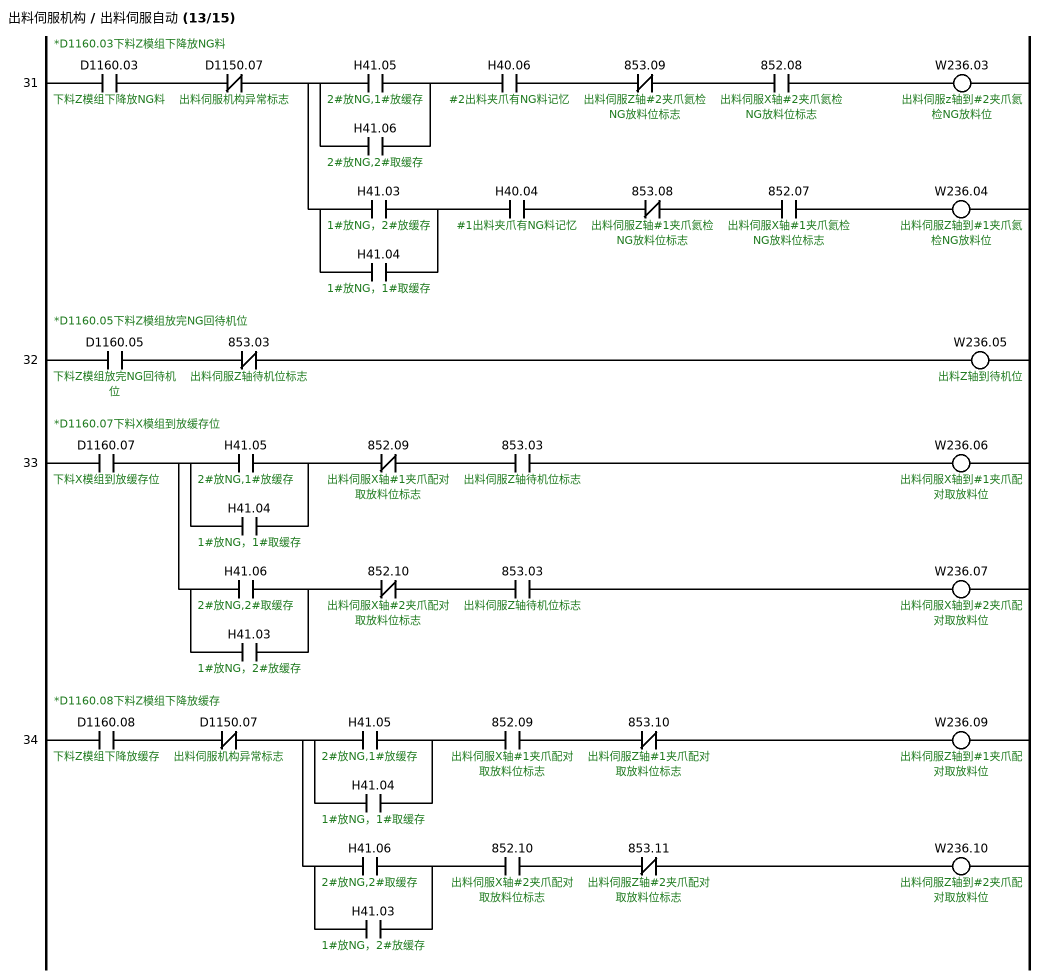
; [picture p456: 出料伺服机构 / 出料伺服自动, rungs 31-34]
; rung 31: *D1160.03下料Z模组下降放NG料
LD D1160.03  ; 下料Z模组下降放NG料
ANDNOT D1150.07  ; 出料伺服机构异常标志
OUT TR0
LD H41.05  ; 2#放NG,1#放缓存
OR H41.06  ; 2#放NG,2#取缓存
ANDLD
AND H40.06  ; #2出料夹爪有NG料记忆
ANDNOT 853.09  ; 出料伺服Z轴#2夹爪氦检NG放料位标志
AND 852.08  ; 出料伺服X轴#2夹爪氦检NG放料位标志
OUT W236.03  ; 出料伺服z轴到#2夹爪氦检NG放料位
LD TR0
LD H41.03  ; 1#放NG，2#放缓存
OR H41.04  ; 1#放NG，1#取缓存
ANDLD
AND H40.04  ; #1出料夹爪有NG料记忆
ANDNOT 853.08  ; 出料伺服Z轴#1夹爪氦检NG放料位标志
AND 852.07  ; 出料伺服X轴#1夹爪氦检NG放料位标志
OUT W236.04  ; 出料伺服Z轴到#1夹爪氦检NG放料位
; rung 32: *D1160.05下料Z模组放完NG回待机位
LD D1160.05  ; 下料Z模组放完NG回待机位
ANDNOT 853.03  ; 出料伺服Z轴待机位标志
OUT W236.05  ; 出料Z轴到待机位
; rung 33: *D1160.07下料X模组到放缓存位
LD D1160.07  ; 下料X模组到放缓存位
OUT TR0
LD H41.05  ; 2#放NG,1#放缓存
OR H41.04  ; 1#放NG，1#取缓存
ANDLD
ANDNOT 852.09  ; 出料伺服X轴#1夹爪配对取放料位标志
AND 853.03  ; 出料伺服Z轴待机位标志
OUT W236.06  ; 出料伺服X轴到#1夹爪配对取放料位
LD TR0
LD H41.06  ; 2#放NG,2#取缓存
OR H41.03  ; 1#放NG，2#放缓存
ANDLD
ANDNOT 852.10  ; 出料伺服X轴#2夹爪配对取放料位标志
AND 853.03  ; 出料伺服Z轴待机位标志
OUT W236.07  ; 出料伺服X轴到#2夹爪配对取放料位
; rung 34: *D1160.08下料Z模组下降放缓存
LD D1160.08  ; 下料Z模组下降放缓存
ANDNOT D1150.07  ; 出料伺服机构异常标志
OUT TR0
LD H41.05  ; 2#放NG,1#放缓存
OR H41.04  ; 1#放NG，1#取缓存
ANDLD
AND 852.09  ; 出料伺服X轴#1夹爪配对取放料位标志
ANDNOT 853.10  ; 出料伺服Z轴#1夹爪配对取放料位标志
OUT W236.09  ; 出料伺服Z轴到#1夹爪配对取放料位
LD TR0
LD H41.06  ; 2#放NG,2#取缓存
OR H41.03  ; 1#放NG，2#放缓存
ANDLD
AND 852.10  ; 出料伺服X轴#2夹爪配对取放料位标志
ANDNOT 853.11  ; 出料伺服Z轴#2夹爪配对取放料位标志
OUT W236.10  ; 出料伺服Z轴到#2夹爪配对取放料位

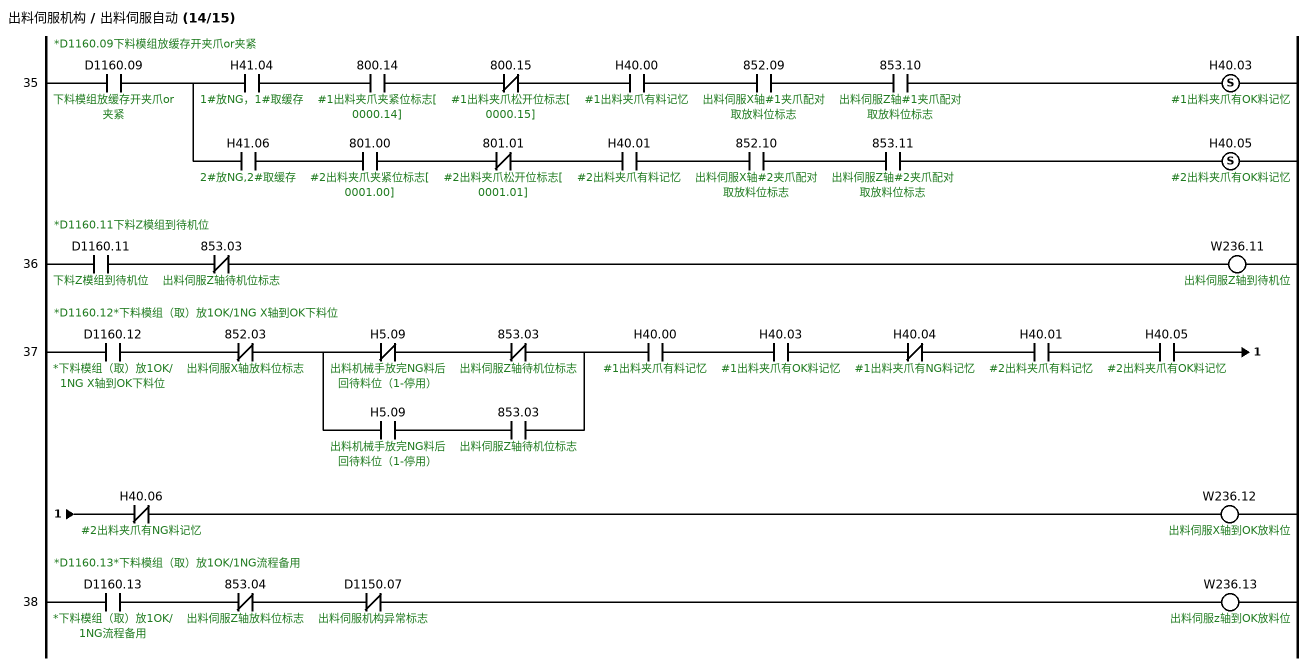
; rung 35: *D1160.09下料模组放缓存开夹爪or夹紧
LD D1160.09  ; 下料模组放缓存开夹爪or夹紧
OUT TR0
AND H41.04  ; 1#放NG，1#取缓存
AND 800.14  ; #1出料夹爪夹紧位标志[0000.14]
ANDNOT 800.15  ; #1出料夹爪松开位标志[0000.15]
AND H40.00  ; #1出料夹爪有料记忆
AND 852.09  ; 出料伺服X轴#1夹爪配对取放料位标志
AND 853.10  ; 出料伺服Z轴#1夹爪配对取放料位标志
SET H40.03  ; #1出料夹爪有OK料记忆
LD TR0
AND H41.06  ; 2#放NG,2#取缓存
AND 801.00  ; #2出料夹爪夹紧位标志[0001.00]
ANDNOT 801.01  ; #2出料夹爪松开位标志[0001.01]
AND H40.01  ; #2出料夹爪有料记忆
AND 852.10  ; 出料伺服X轴#2夹爪配对取放料位标志
AND 853.11  ; 出料伺服Z轴#2夹爪配对取放料位标志
SET H40.05  ; #2出料夹爪有OK料记忆
; rung 36: *D1160.11下料Z模组到待机位
LD D1160.11  ; 下料Z模组到待机位
ANDNOT 853.03  ; 出料伺服Z轴待机位标志
OUT W236.11  ; 出料伺服Z轴到待机位
; rung 37: *D1160.12*下料模组（取）放1OK/1NG X轴到OK下料位
LD D1160.12  ; *下料模组（取）放1OK/1NG X轴到OK下料位
ANDNOT 852.03  ; 出料伺服X轴放料位标志
LDNOT H5.09  ; 出料机械手放完NG料后回待料位（1-停用）
ANDNOT 853.03  ; 出料伺服Z轴待机位标志  // X轴移动条件必须是Z轴在安全位（20190417）
LD H5.09  ; 出料机械手放完NG料后回待料位（1-停用）
AND 853.03  ; 出料伺服Z轴待机位标志
ORLD
ANDLD
AND H40.00  ; #1出料夹爪有料记忆
AND H40.03  ; #1出料夹爪有OK料记忆
ANDNOT H40.04  ; #1出料夹爪有NG料记忆
AND H40.01  ; #2出料夹爪有料记忆
AND H40.05  ; #2出料夹爪有OK料记忆
ANDNOT H40.06  ; #2出料夹爪有NG料记忆
OUT W236.12  ; 出料伺服X轴到OK放料位
; rung 38: *D1160.13*下料模组（取）放1OK/1NG流程备用
LD D1160.13  ; *下料模组（取）放1OK/1NG流程备用
ANDNOT 853.04  ; 出料伺服Z轴放料位标志
ANDNOT D1150.07  ; 出料伺服机构异常标志
OUT W236.13  ; 出料伺服z轴到OK放料位

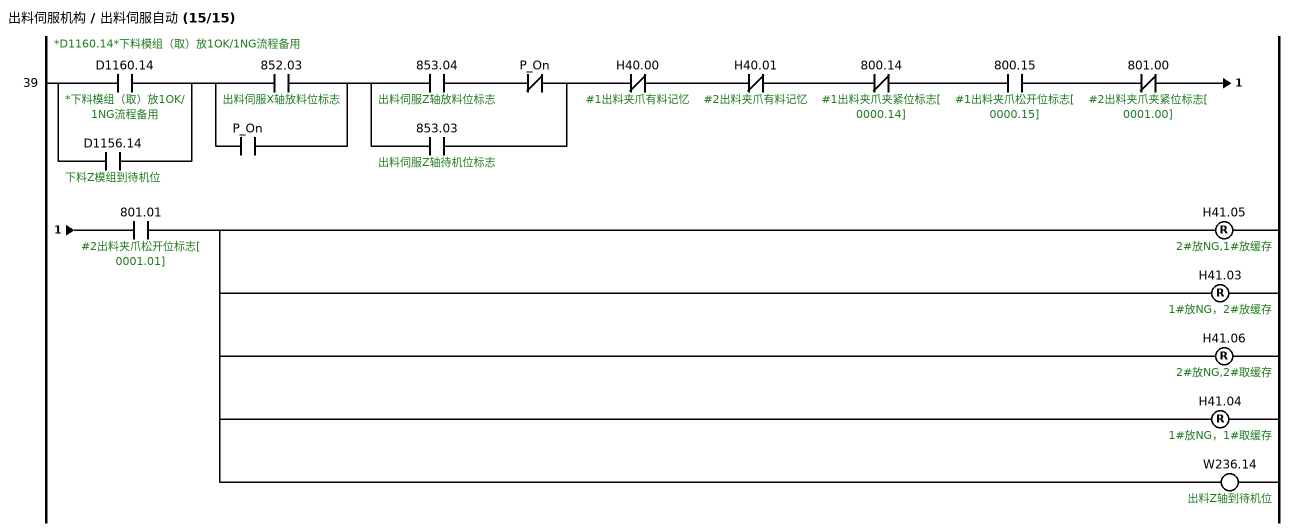
; rung 39: *D1160.14*下料模组（取）放1OK/1NG流程备用
LD D1160.14  ; *下料模组（取）放1OK/1NG流程备用
OR D1156.14  ; 下料Z模组到待机位
LD 852.03  ; 出料伺服X轴放料位标志
OR P_On
ANDLD
LD 853.04  ; 出料伺服Z轴放料位标志
ANDNOT P_On
OR 853.03  ; 出料伺服Z轴待机位标志
ANDLD
ANDNOT H40.00  ; #1出料夹爪有料记忆
ANDNOT H40.01  ; #2出料夹爪有料记忆
ANDNOT 800.14  ; #1出料夹爪夹紧位标志[0000.14]
AND 800.15  ; #1出料夹爪松开位标志[0000.15]
ANDNOT 801.00  ; #2出料夹爪夹紧位标志[0001.00]
AND 801.01  ; #2出料夹爪松开位标志[0001.01]
RSET H41.05  ; 2#放NG,1#放缓存
RSET H41.03  ; 1#放NG，2#放缓存
RSET H41.06  ; 2#放NG,2#取缓存
RSET H41.04  ; 1#放NG，1#取缓存
OUT W236.14  ; 出料Z轴到待机位

### Section 工站复位

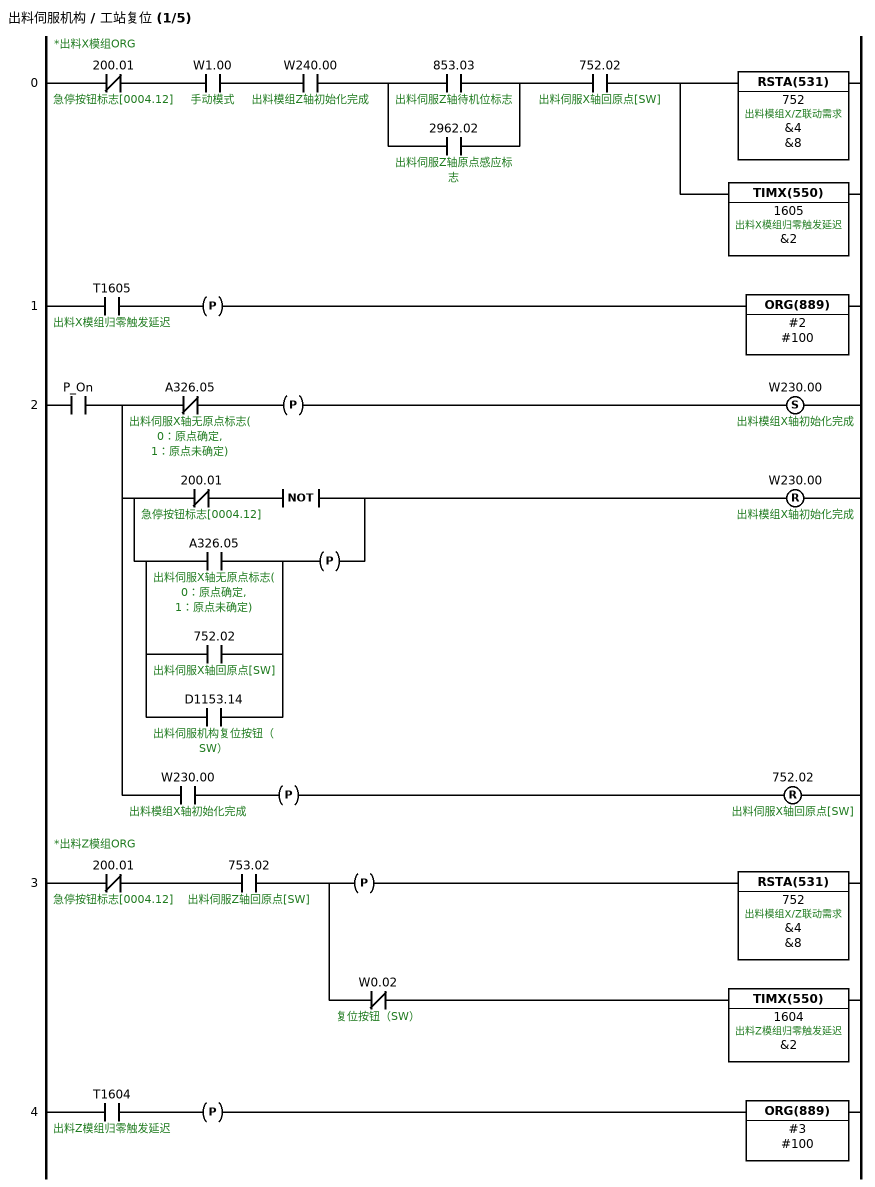
; rung 0: *出料X模组ORG
LDNOT 200.01  ; 急停按钮标志[0004.12]
AND W1.00  ; 手动模式
AND W240.00  ; 出料模组Z轴初始化完成
LD 853.03  ; 出料伺服Z轴待机位标志
OR 2962.02  ; 出料伺服Z轴原点感应标志
ANDLD
AND 752.02  ; 出料伺服X轴回原点[SW]
RSTA(531) 752 &4 &8  ; 出料模组X/Z联动需求
TIMX(550) 1605 &2  ; 出料X模组归零触发延迟
; rung 1
LD T1605  ; 出料X模组归零触发延迟
UP(521)
ORG(889) #2 #100
; rung 2
LD P_On
OUT TR0
ANDNOT A326.05  ; 出料伺服X轴无原点标志(0：原点确定,1：原点未确定)
UP(521)
SET W230.00  ; 出料模组X轴初始化完成
LD TR0
LDNOT 200.01  ; 急停按钮标志[0004.12]
NOT(520)
LD A326.05  ; 出料伺服X轴无原点标志(0：原点确定,1：原点未确定)
OR 752.02  ; 出料伺服X轴回原点[SW]
OR D1153.14  ; 出料伺服机构复位按钮（SW）
UP(521)
ORLD
ANDLD
RSET W230.00  ; 出料模组X轴初始化完成
LD TR0
AND W230.00  ; 出料模组X轴初始化完成
UP(521)
RSET 752.02  ; 出料伺服X轴回原点[SW]
; rung 3: *出料Z模组ORG
LDNOT 200.01  ; 急停按钮标志[0004.12]
AND 753.02  ; 出料伺服Z轴回原点[SW]
OUT TR0
UP(521)
RSTA(531) 752 &4 &8  ; 出料模组X/Z联动需求
LD TR0
ANDNOT W0.02  ; 复位按钮（SW）
TIMX(550) 1604 &2  ; 出料Z模组归零触发延迟
; rung 4
LD T1604  ; 出料Z模组归零触发延迟
UP(521)
ORG(889) #3 #100

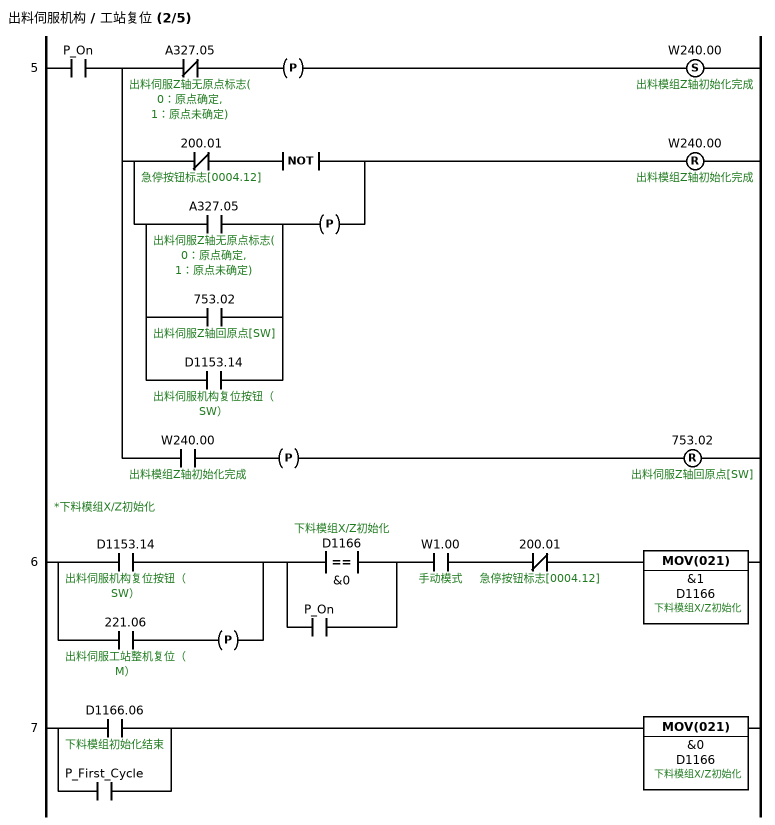
; rung 5
LD P_On
OUT TR0
ANDNOT A327.05  ; 出料伺服Z轴无原点标志(0：原点确定,1：原点未确定)
UP(521)
SET W240.00  ; 出料模组Z轴初始化完成
LD TR0
LDNOT 200.01  ; 急停按钮标志[0004.12]
NOT(520)
LD A327.05  ; 出料伺服Z轴无原点标志(0：原点确定,1：原点未确定)
OR 753.02  ; 出料伺服Z轴回原点[SW]
OR D1153.14  ; 出料伺服机构复位按钮（SW）
UP(521)
ORLD
ANDLD
RSET W240.00  ; 出料模组Z轴初始化完成
LD TR0
AND W240.00  ; 出料模组Z轴初始化完成
UP(521)
RSET 753.02  ; 出料伺服Z轴回原点[SW]
; rung 6: *下料模组X/Z初始化
LD D1153.14  ; 出料伺服机构复位按钮（SW）
LD 221.06  ; 出料伺服工站整机复位（M）
UP(521)
ORLD
LD=(300) D1166 &0  ; 下料模组X/Z初始化
OR P_On
ANDLD
AND W1.00  ; 手动模式
ANDNOT 200.01  ; 急停按钮标志[0004.12]
MOV(021) &1 D1166  ; 下料模组X/Z初始化
; rung 7
LD D1166.06  ; 下料模组初始化结束
OR P_First_Cycle
MOV(021) &0 D1166  ; 下料模组X/Z初始化

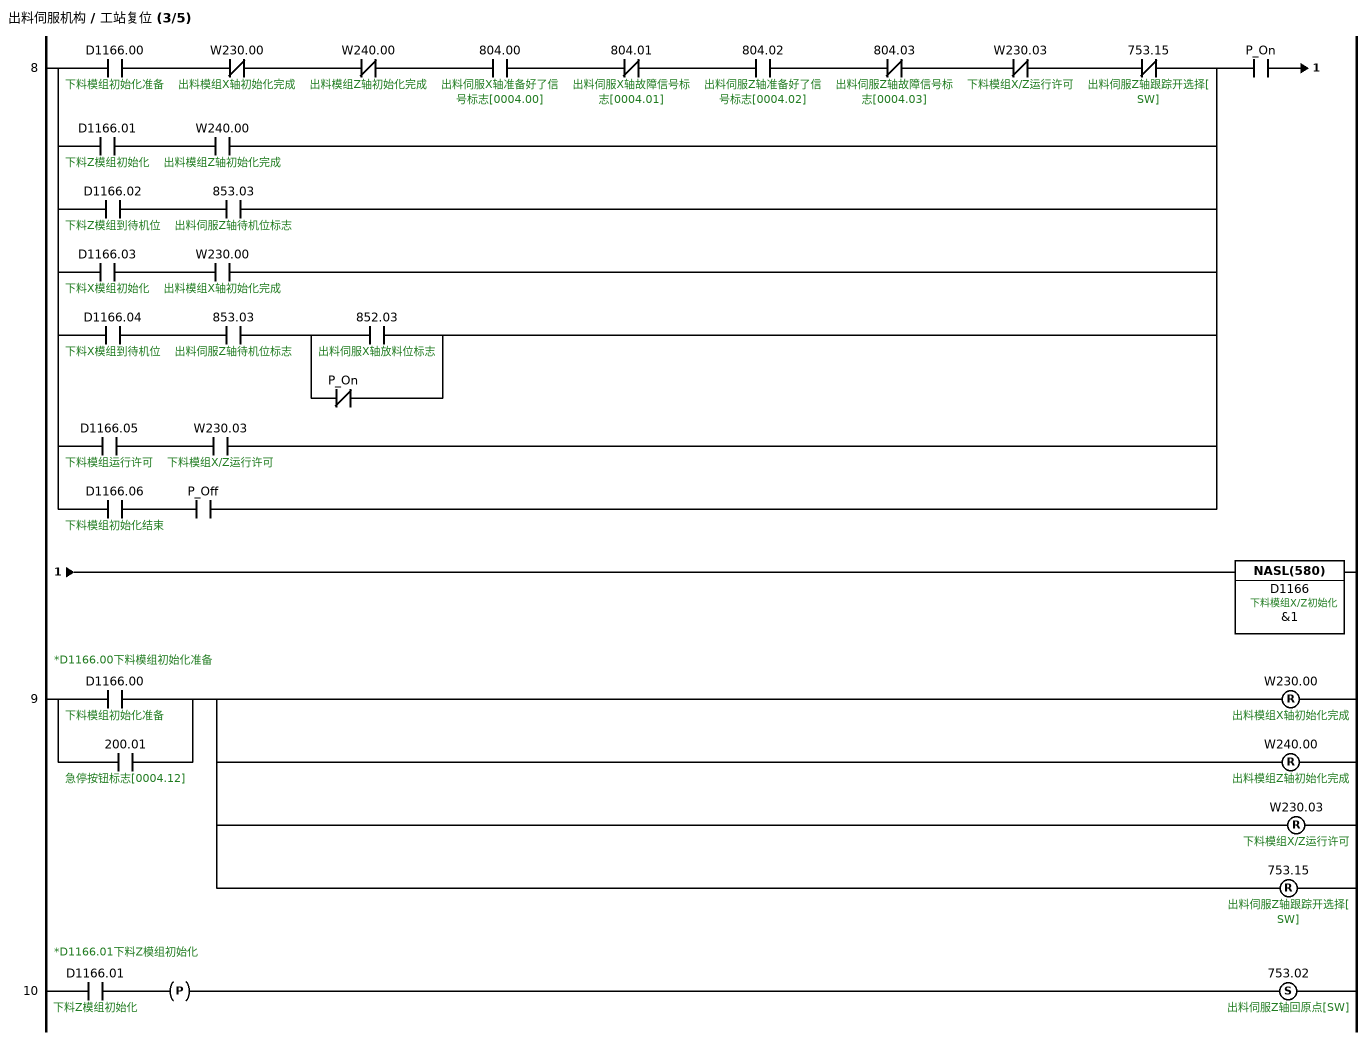
; rung 8
LD D1166.00  ; 下料模组初始化准备
ANDNOT W230.00  ; 出料模组X轴初始化完成
ANDNOT W240.00  ; 出料模组Z轴初始化完成
AND 804.00  ; 出料伺服X轴准备好了信号标志[0004.00]
ANDNOT 804.01  ; 出料伺服X轴故障信号标志[0004.01]
AND 804.02  ; 出料伺服Z轴准备好了信号标志[0004.02]
ANDNOT 804.03  ; 出料伺服Z轴故障信号标志[0004.03]
ANDNOT W230.03  ; 下料模组X/Z运行许可
ANDNOT 753.15  ; 出料伺服Z轴跟踪开选择[SW]
LD D1166.01  ; 下料Z模组初始化
AND W240.00  ; 出料模组Z轴初始化完成
ORLD
LD D1166.02  ; 下料Z模组到待机位
AND 853.03  ; 出料伺服Z轴待机位标志
ORLD
LD D1166.03  ; 下料X模组初始化
AND W230.00  ; 出料模组X轴初始化完成
ORLD
LD D1166.04  ; 下料X模组到待机位
AND 853.03  ; 出料伺服Z轴待机位标志
LD 852.03  ; 出料伺服X轴放料位标志
ORNOT P_On
ANDLD
ORLD
LD D1166.05  ; 下料模组运行许可
AND W230.03  ; 下料模组X/Z运行许可
ORLD
LD D1166.06  ; 下料模组初始化结束
AND P_Off
ORLD
AND P_On
NASL(580) D1166 &1  ; 下料模组X/Z初始化
; rung 9: *D1166.00下料模组初始化准备
LD D1166.00  ; 下料模组初始化准备
OR 200.01  ; 急停按钮标志[0004.12]
RSET W230.00  ; 出料模组X轴初始化完成
RSET W240.00  ; 出料模组Z轴初始化完成
RSET W230.03  ; 下料模组X/Z运行许可
RSET 753.15  ; 出料伺服Z轴跟踪开选择[SW]
; rung 10: *D1166.01下料Z模组初始化
LD D1166.01  ; 下料Z模组初始化
UP(521)
SET 753.02  ; 出料伺服Z轴回原点[SW]

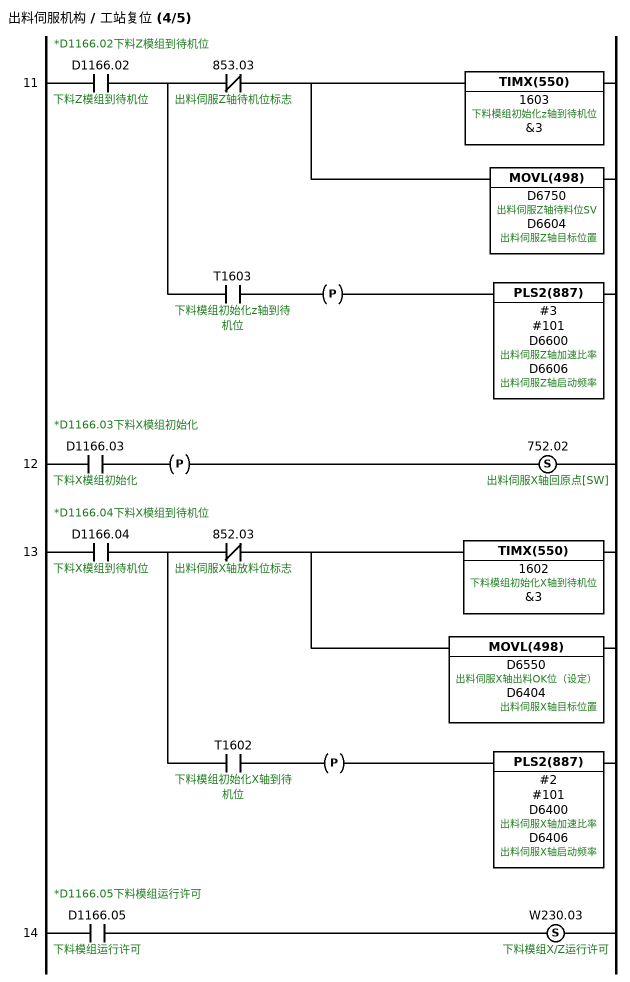
; rung 11: *D1166.02下料Z模组到待机位
LD D1166.02  ; 下料Z模组到待机位
OUT TR0
ANDNOT 853.03  ; 出料伺服Z轴待机位标志
TIMX(550) 1603 &3  ; 下料模组初始化z轴到待机位
MOVL(498) D6750 D6604  ; 出料伺服Z轴待料位SV, 出料伺服Z轴目标位置
LD TR0
AND T1603  ; 下料模组初始化z轴到待机位
UP(521)
PLS2(887) #3 #101 D6600 D6606  ; 出料伺服Z轴加速比率, 出料伺服Z轴启动频率
; rung 12: *D1166.03下料X模组初始化
LD D1166.03  ; 下料X模组初始化
UP(521)
SET 752.02  ; 出料伺服X轴回原点[SW]
; rung 13: *D1166.04下料X模组到待机位
LD D1166.04  ; 下料X模组到待机位
OUT TR0
ANDNOT 852.03  ; 出料伺服X轴放料位标志
TIMX(550) 1602 &3  ; 下料模组初始化X轴到待机位
MOVL(498) D6550 D6404  ; 出料伺服X轴出料OK位（设定）, 出料伺服X轴目标位置
LD TR0
AND T1602  ; 下料模组初始化X轴到待机位
UP(521)
PLS2(887) #2 #101 D6400 D6406  ; 出料伺服X轴加速比率, 出料伺服X轴启动频率
; rung 14: *D1166.05下料模组运行许可
LD D1166.05  ; 下料模组运行许可
SET W230.03  ; 下料模组X/Z运行许可

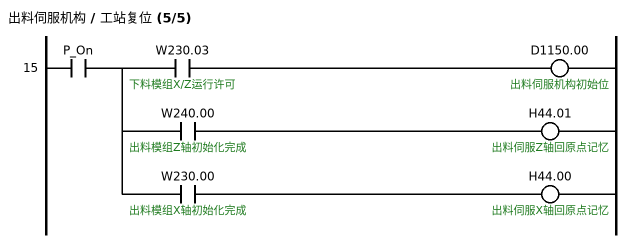
; rung 15
LD P_On
OUT TR0
AND W230.03  ; 下料模组X/Z运行许可
OUT D1150.00  ; 出料伺服机构初始位
LD TR0
AND W240.00  ; 出料模组Z轴初始化完成
OUT H44.01  ; 出料伺服Z轴回原点记忆
LD TR0
AND W230.00  ; 出料模组X轴初始化完成
OUT H44.00  ; 出料伺服X轴回原点记忆

### Section 指示灯

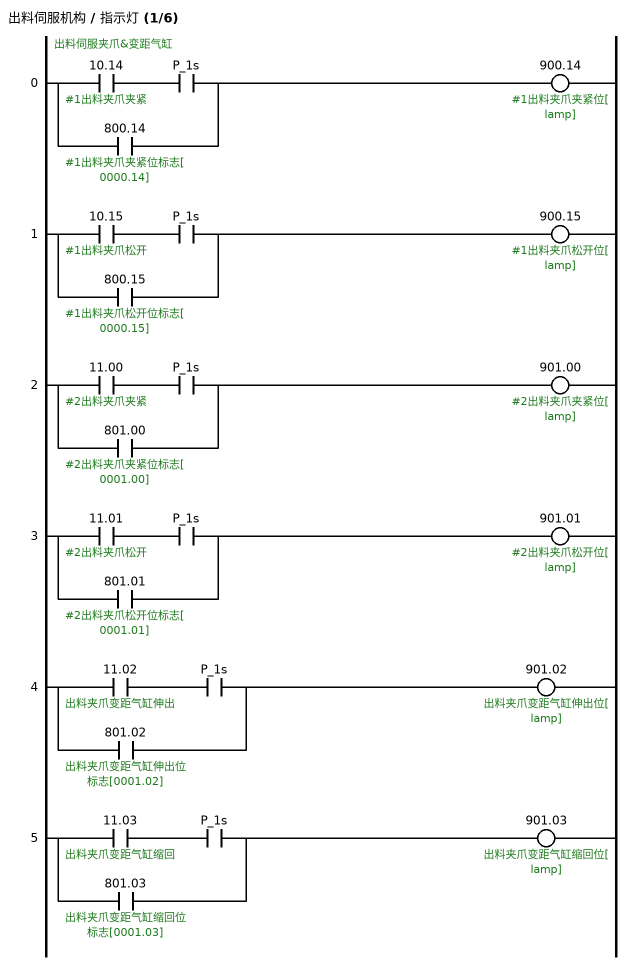
; rung 0: 出料伺服夹爪&变距气缸
LD 10.14  ; #1出料夹爪夹紧
AND P_1s
OR 800.14  ; #1出料夹爪夹紧位标志[0000.14]
OUT 900.14  ; #1出料夹爪夹紧位[lamp]
; rung 1
LD 10.15  ; #1出料夹爪松开
AND P_1s
OR 800.15  ; #1出料夹爪松开位标志[0000.15]
OUT 900.15  ; #1出料夹爪松开位[lamp]
; rung 2
LD 11.00  ; #2出料夹爪夹紧
AND P_1s
OR 801.00  ; #2出料夹爪夹紧位标志[0001.00]
OUT 901.00  ; #2出料夹爪夹紧位[lamp]
; rung 3
LD 11.01  ; #2出料夹爪松开
AND P_1s
OR 801.01  ; #2出料夹爪松开位标志[0001.01]
OUT 901.01  ; #2出料夹爪松开位[lamp]
; rung 4
LD 11.02  ; 出料夹爪变距气缸伸出
AND P_1s
OR 801.02  ; 出料夹爪变距气缸伸出位标志[0001.02]
OUT 901.02  ; 出料夹爪变距气缸伸出位[lamp]
; rung 5
LD 11.03  ; 出料夹爪变距气缸缩回
AND P_1s
OR 801.03  ; 出料夹爪变距气缸缩回位标志[0001.03]
OUT 901.03  ; 出料夹爪变距气缸缩回位[lamp]

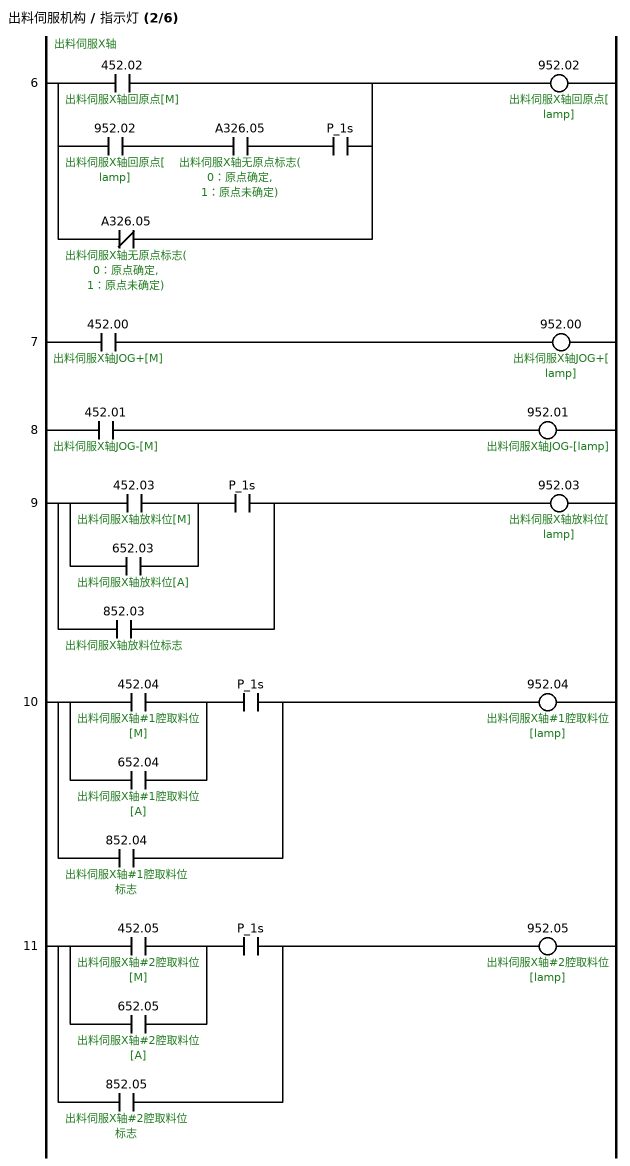
; rung 6: 出料伺服X轴
LD 452.02  ; 出料伺服X轴回原点[M]
LD 952.02  ; 出料伺服X轴回原点[lamp]
AND A326.05  ; 出料伺服X轴无原点标志(0：原点确定,1：原点未确定)
AND P_1s
ORLD
ORNOT A326.05  ; 出料伺服X轴无原点标志(0：原点确定,1：原点未确定)
OUT 952.02  ; 出料伺服X轴回原点[lamp]
; rung 7
LD 452.00  ; 出料伺服X轴JOG+[M]
OUT 952.00  ; 出料伺服X轴JOG+[lamp]
; rung 8
LD 452.01  ; 出料伺服X轴JOG-[M]
OUT 952.01  ; 出料伺服X轴JOG-[lamp]
; rung 9
LD 452.03  ; 出料伺服X轴放料位[M]
OR 652.03  ; 出料伺服X轴放料位[A]
AND P_1s
OR 852.03  ; 出料伺服X轴放料位标志
OUT 952.03  ; 出料伺服X轴放料位[lamp]
; rung 10
LD 452.04  ; 出料伺服X轴#1腔取料位[M]
OR 652.04  ; 出料伺服X轴#1腔取料位[A]
AND P_1s
OR 852.04  ; 出料伺服X轴#1腔取料位标志
OUT 952.04  ; 出料伺服X轴#1腔取料位[lamp]
; rung 11
LD 452.05  ; 出料伺服X轴#2腔取料位[M]
OR 652.05  ; 出料伺服X轴#2腔取料位[A]
AND P_1s
OR 852.05  ; 出料伺服X轴#2腔取料位标志
OUT 952.05  ; 出料伺服X轴#2腔取料位[lamp]

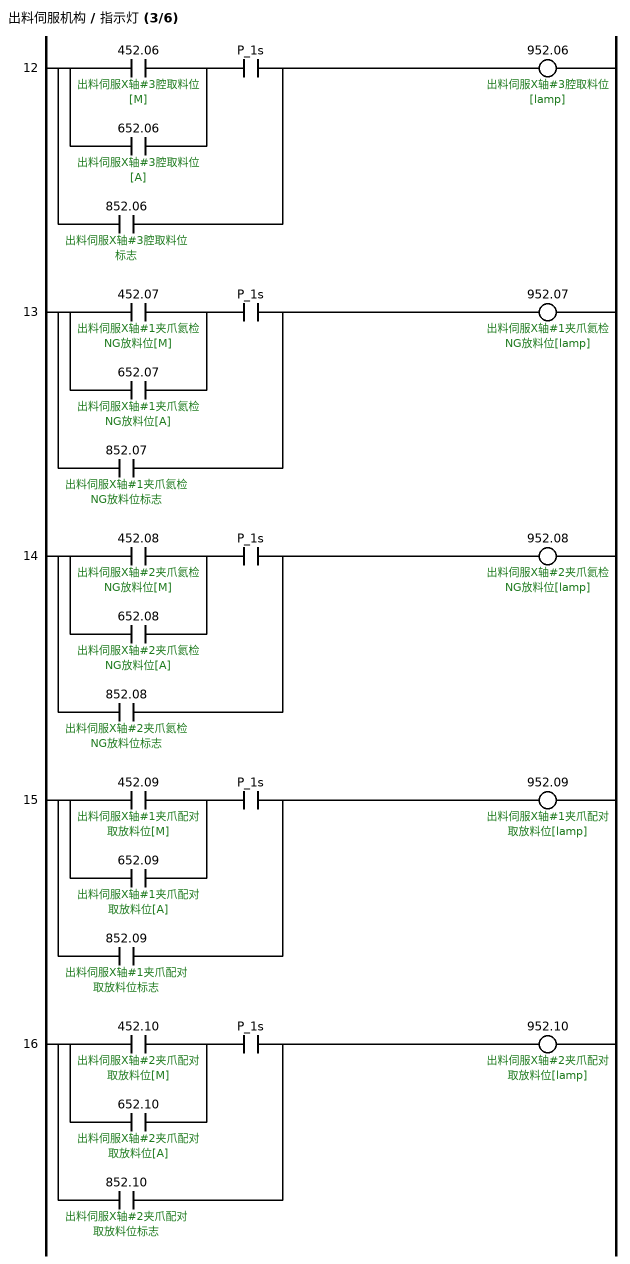
; rung 12
LD 452.06  ; 出料伺服X轴#3腔取料位[M]
OR 652.06  ; 出料伺服X轴#3腔取料位[A]
AND P_1s
OR 852.06  ; 出料伺服X轴#3腔取料位标志
OUT 952.06  ; 出料伺服X轴#3腔取料位[lamp]
; rung 13
LD 452.07  ; 出料伺服X轴#1夹爪氦检NG放料位[M]
OR 652.07  ; 出料伺服X轴#1夹爪氦检NG放料位[A]
AND P_1s
OR 852.07  ; 出料伺服X轴#1夹爪氦检NG放料位标志
OUT 952.07  ; 出料伺服X轴#1夹爪氦检NG放料位[lamp]
; rung 14
LD 452.08  ; 出料伺服X轴#2夹爪氦检NG放料位[M]
OR 652.08  ; 出料伺服X轴#2夹爪氦检NG放料位[A]
AND P_1s
OR 852.08  ; 出料伺服X轴#2夹爪氦检NG放料位标志
OUT 952.08  ; 出料伺服X轴#2夹爪氦检NG放料位[lamp]
; rung 15
LD 452.09  ; 出料伺服X轴#1夹爪配对取放料位[M]
OR 652.09  ; 出料伺服X轴#1夹爪配对取放料位[A]
AND P_1s
OR 852.09  ; 出料伺服X轴#1夹爪配对取放料位标志
OUT 952.09  ; 出料伺服X轴#1夹爪配对取放料位[lamp]
; rung 16
LD 452.10  ; 出料伺服X轴#2夹爪配对取放料位[M]
OR 652.10  ; 出料伺服X轴#2夹爪配对取放料位[A]
AND P_1s
OR 852.10  ; 出料伺服X轴#2夹爪配对取放料位标志
OUT 952.10  ; 出料伺服X轴#2夹爪配对取放料位[lamp]

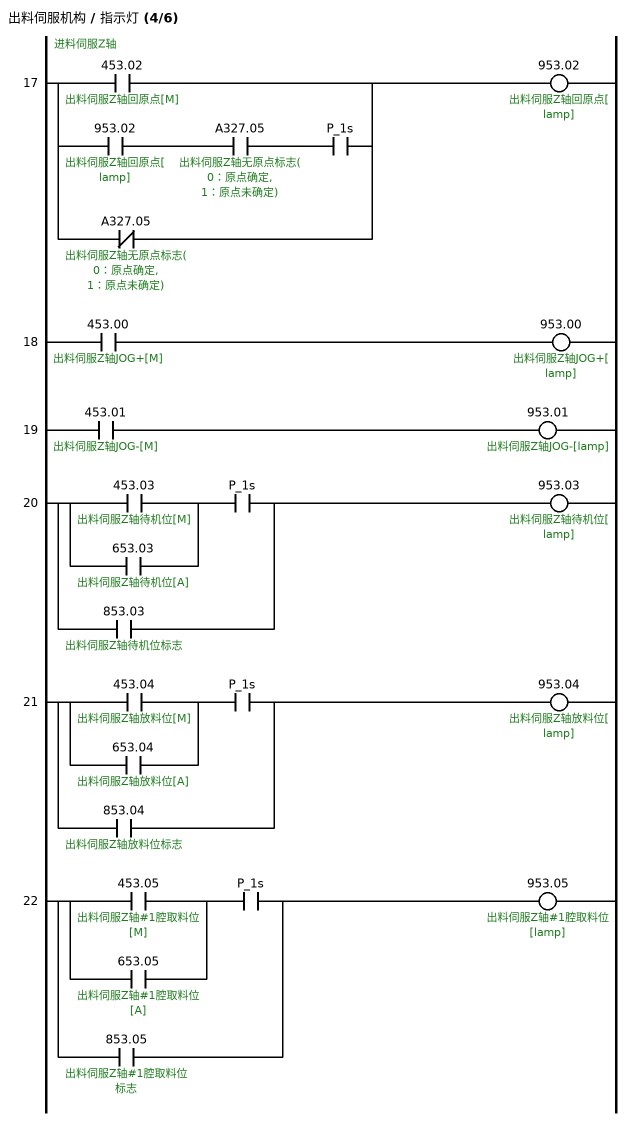
; rung 17: 进料伺服Z轴
LD 453.02  ; 出料伺服Z轴回原点[M]
LD 953.02  ; 出料伺服Z轴回原点[lamp]
AND A327.05  ; 出料伺服Z轴无原点标志(0：原点确定,1：原点未确定)
AND P_1s
ORLD
ORNOT A327.05  ; 出料伺服Z轴无原点标志(0：原点确定,1：原点未确定)
OUT 953.02  ; 出料伺服Z轴回原点[lamp]
; rung 18
LD 453.00  ; 出料伺服Z轴JOG+[M]
OUT 953.00  ; 出料伺服Z轴JOG+[lamp]
; rung 19
LD 453.01  ; 出料伺服Z轴JOG-[M]
OUT 953.01  ; 出料伺服Z轴JOG-[lamp]
; rung 20
LD 453.03  ; 出料伺服Z轴待机位[M]
OR 653.03  ; 出料伺服Z轴待机位[A]
AND P_1s
OR 853.03  ; 出料伺服Z轴待机位标志
OUT 953.03  ; 出料伺服Z轴待机位[lamp]
; rung 21
LD 453.04  ; 出料伺服Z轴放料位[M]
OR 653.04  ; 出料伺服Z轴放料位[A]
AND P_1s
OR 853.04  ; 出料伺服Z轴放料位标志
OUT 953.04  ; 出料伺服Z轴放料位[lamp]
; rung 22
LD 453.05  ; 出料伺服Z轴#1腔取料位[M]
OR 653.05  ; 出料伺服Z轴#1腔取料位[A]
AND P_1s
OR 853.05  ; 出料伺服Z轴#1腔取料位标志
OUT 953.05  ; 出料伺服Z轴#1腔取料位[lamp]

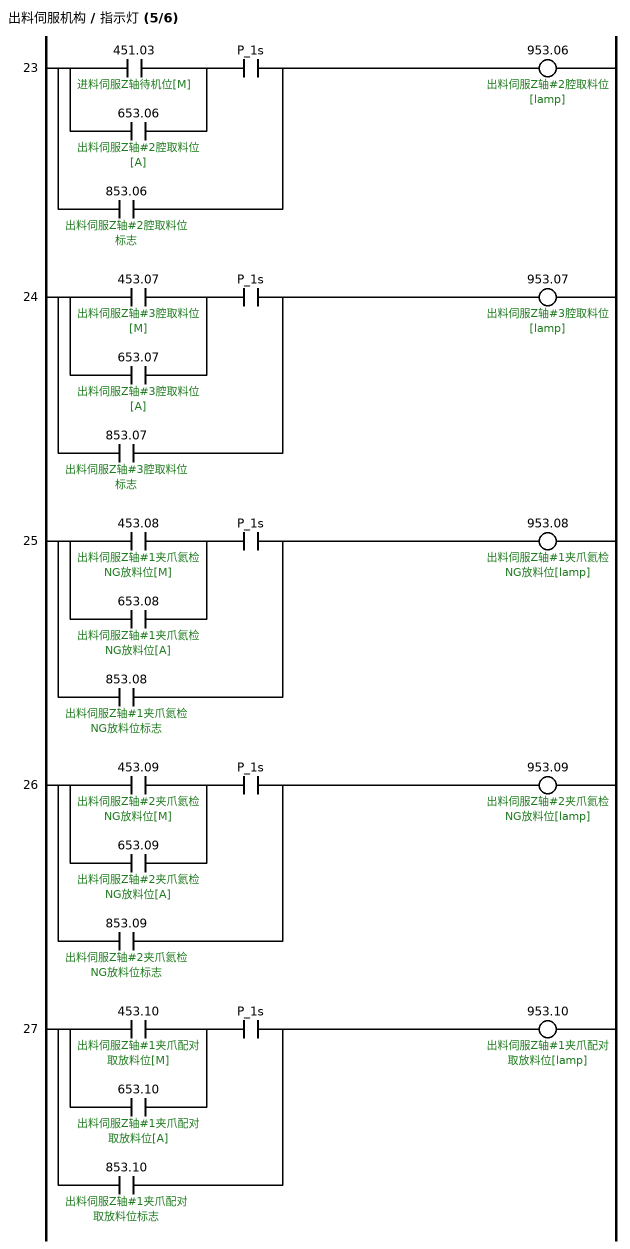
; rung 23
LD 451.03  ; 进料伺服Z轴待机位[M]
OR 653.06  ; 出料伺服Z轴#2腔取料位[A]
AND P_1s
OR 853.06  ; 出料伺服Z轴#2腔取料位标志
OUT 953.06  ; 出料伺服Z轴#2腔取料位[lamp]
; rung 24
LD 453.07  ; 出料伺服Z轴#3腔取料位[M]
OR 653.07  ; 出料伺服Z轴#3腔取料位[A]
AND P_1s
OR 853.07  ; 出料伺服Z轴#3腔取料位标志
OUT 953.07  ; 出料伺服Z轴#3腔取料位[lamp]
; rung 25
LD 453.08  ; 出料伺服Z轴#1夹爪氦检NG放料位[M]
OR 653.08  ; 出料伺服Z轴#1夹爪氦检NG放料位[A]
AND P_1s
OR 853.08  ; 出料伺服Z轴#1夹爪氦检NG放料位标志
OUT 953.08  ; 出料伺服Z轴#1夹爪氦检NG放料位[lamp]
; rung 26
LD 453.09  ; 出料伺服Z轴#2夹爪氦检NG放料位[M]
OR 653.09  ; 出料伺服Z轴#2夹爪氦检NG放料位[A]
AND P_1s
OR 853.09  ; 出料伺服Z轴#2夹爪氦检NG放料位标志
OUT 953.09  ; 出料伺服Z轴#2夹爪氦检NG放料位[lamp]
; rung 27
LD 453.10  ; 出料伺服Z轴#1夹爪配对取放料位[M]
OR 653.10  ; 出料伺服Z轴#1夹爪配对取放料位[A]
AND P_1s
OR 853.10  ; 出料伺服Z轴#1夹爪配对取放料位标志
OUT 953.10  ; 出料伺服Z轴#1夹爪配对取放料位[lamp]

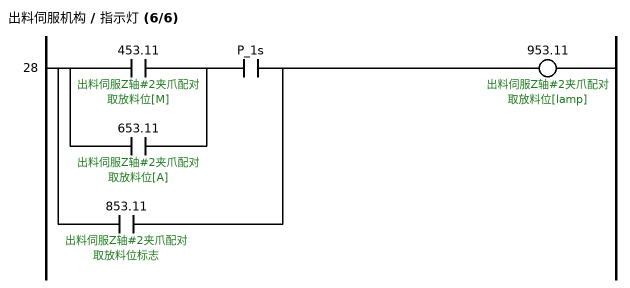
; rung 28
LD 453.11  ; 出料伺服Z轴#2夹爪配对取放料位[M]
OR 653.11  ; 出料伺服Z轴#2夹爪配对取放料位[A]
AND P_1s
OR 853.11  ; 出料伺服Z轴#2夹爪配对取放料位标志
OUT 953.11  ; 出料伺服Z轴#2夹爪配对取放料位[lamp]

### Section 外部输出

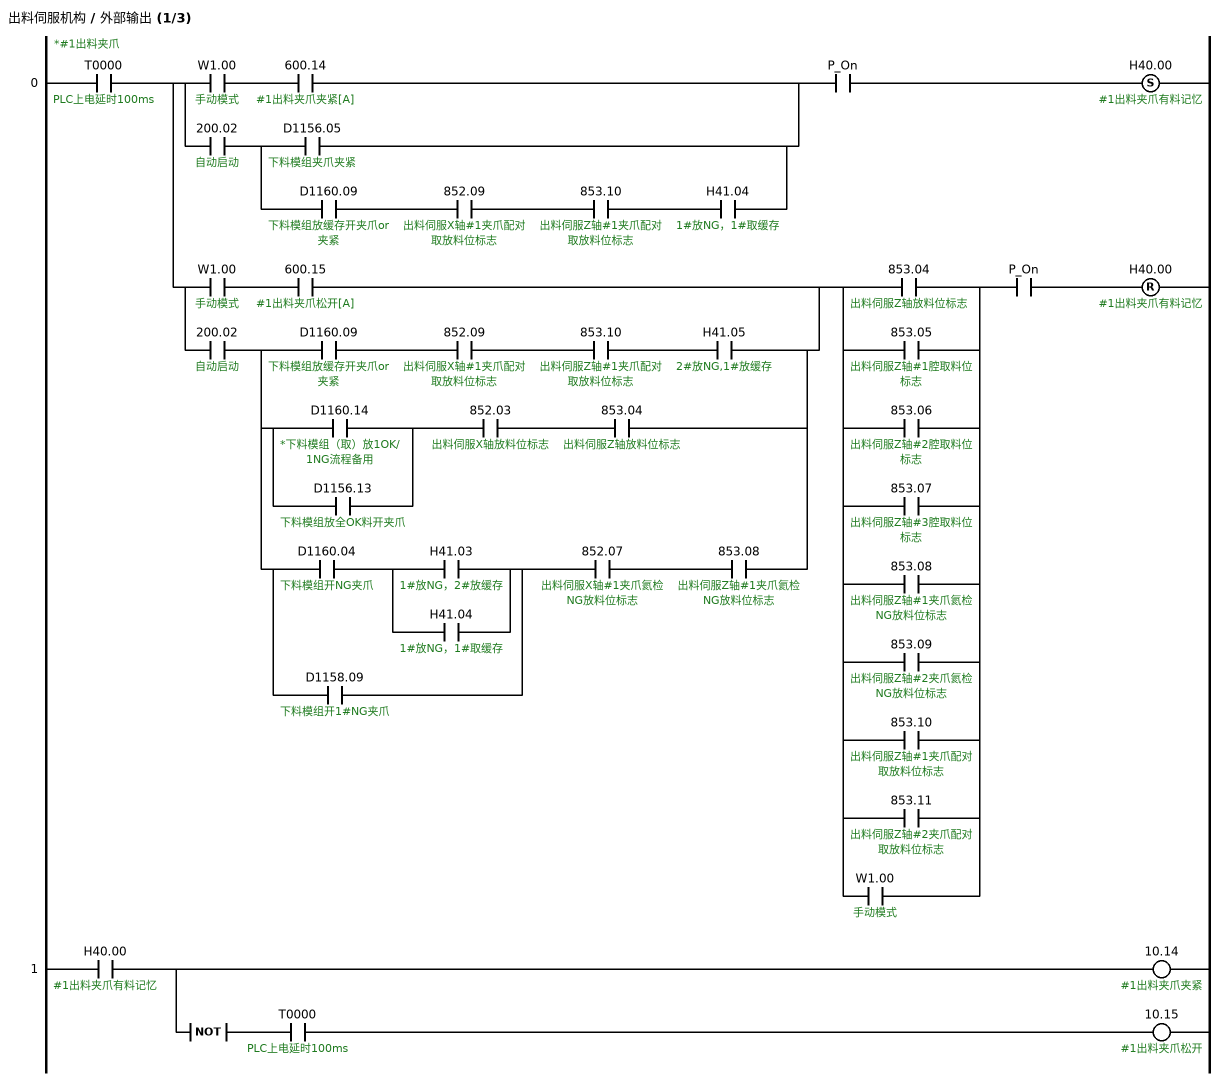
; rung 0: *#1出料夹爪
LD T0000  ; PLC上电延时100ms
OUT TR0
LD W1.00  ; 手动模式
AND 600.14  ; #1出料夹爪夹紧[A]
LD 200.02  ; 自动启动
LD D1156.05  ; 下料模组夹爪夹紧
LD D1160.09  ; 下料模组放缓存开夹爪or夹紧
AND 852.09  ; 出料伺服X轴#1夹爪配对取放料位标志
AND 853.10  ; 出料伺服Z轴#1夹爪配对取放料位标志
AND H41.04  ; 1#放NG，1#取缓存
ORLD
ANDLD
ORLD
ANDLD
AND P_On
SET H40.00  ; #1出料夹爪有料记忆
LD TR0
LD W1.00  ; 手动模式
AND 600.15  ; #1出料夹爪松开[A]
LD 200.02  ; 自动启动
LD D1160.09  ; 下料模组放缓存开夹爪or夹紧
AND 852.09  ; 出料伺服X轴#1夹爪配对取放料位标志
AND 853.10  ; 出料伺服Z轴#1夹爪配对取放料位标志
AND H41.05  ; 2#放NG,1#放缓存
LD D1160.14  ; *下料模组（取）放1OK/1NG流程备用
OR D1156.13  ; 下料模组放全OK料开夹爪
AND 852.03  ; 出料伺服X轴放料位标志
AND 853.04  ; 出料伺服Z轴放料位标志
ORLD
LD D1160.04  ; 下料模组开NG夹爪
LD H41.03  ; 1#放NG，2#放缓存
OR H41.04  ; 1#放NG，1#取缓存
ANDLD
OR D1158.09  ; 下料模组开1#NG夹爪
AND 852.07  ; 出料伺服X轴#1夹爪氦检NG放料位标志
AND 853.08  ; 出料伺服Z轴#1夹爪氦检NG放料位标志
ORLD
ANDLD
ORLD
ANDLD
LD 853.04  ; 出料伺服Z轴放料位标志
OR 853.05  ; 出料伺服Z轴#1腔取料位标志
OR 853.06  ; 出料伺服Z轴#2腔取料位标志
OR 853.07  ; 出料伺服Z轴#3腔取料位标志
OR 853.08  ; 出料伺服Z轴#1夹爪氦检NG放料位标志
OR 853.09  ; 出料伺服Z轴#2夹爪氦检NG放料位标志
OR 853.10  ; 出料伺服Z轴#1夹爪配对取放料位标志
OR 853.11  ; 出料伺服Z轴#2夹爪配对取放料位标志
OR W1.00  ; 手动模式
ANDLD
AND P_On
RSET H40.00  ; #1出料夹爪有料记忆
; rung 1
LD H40.00  ; #1出料夹爪有料记忆
OUT 10.14  ; #1出料夹爪夹紧
NOT(520)
AND T0000  ; PLC上电延时100ms
OUT 10.15  ; #1出料夹爪松开

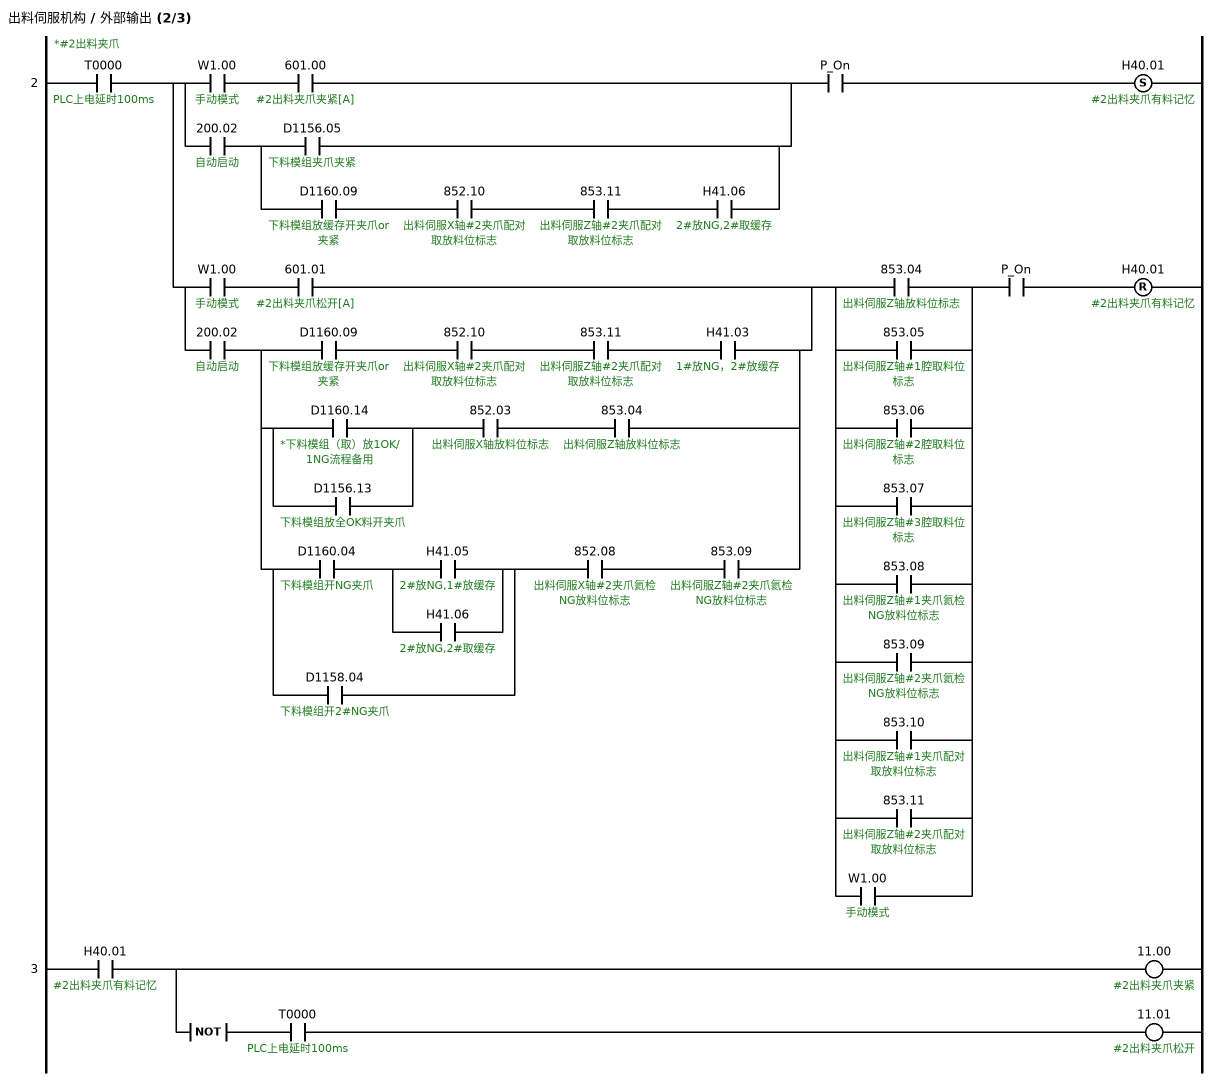
; rung 2: *#2出料夹爪
LD T0000  ; PLC上电延时100ms
OUT TR0
LD W1.00  ; 手动模式
AND 601.00  ; #2出料夹爪夹紧[A]
LD 200.02  ; 自动启动
LD D1156.05  ; 下料模组夹爪夹紧
LD D1160.09  ; 下料模组放缓存开夹爪or夹紧
AND 852.10  ; 出料伺服X轴#2夹爪配对取放料位标志
AND 853.11  ; 出料伺服Z轴#2夹爪配对取放料位标志
AND H41.06  ; 2#放NG,2#取缓存
ORLD
ANDLD
ORLD
ANDLD
AND P_On
SET H40.01  ; #2出料夹爪有料记忆
LD TR0
LD W1.00  ; 手动模式
AND 601.01  ; #2出料夹爪松开[A]
LD 200.02  ; 自动启动
LD D1160.09  ; 下料模组放缓存开夹爪or夹紧
AND 852.10  ; 出料伺服X轴#2夹爪配对取放料位标志
AND 853.11  ; 出料伺服Z轴#2夹爪配对取放料位标志
AND H41.03  ; 1#放NG，2#放缓存
LD D1160.14  ; *下料模组（取）放1OK/1NG流程备用
OR D1156.13  ; 下料模组放全OK料开夹爪
AND 852.03  ; 出料伺服X轴放料位标志
AND 853.04  ; 出料伺服Z轴放料位标志
ORLD
LD D1160.04  ; 下料模组开NG夹爪
LD H41.05  ; 2#放NG,1#放缓存
OR H41.06  ; 2#放NG,2#取缓存
ANDLD
OR D1158.04  ; 下料模组开2#NG夹爪
AND 852.08  ; 出料伺服X轴#2夹爪氦检NG放料位标志
AND 853.09  ; 出料伺服Z轴#2夹爪氦检NG放料位标志
ORLD
ANDLD
ORLD
ANDLD
LD 853.04  ; 出料伺服Z轴放料位标志
OR 853.05  ; 出料伺服Z轴#1腔取料位标志
OR 853.06  ; 出料伺服Z轴#2腔取料位标志
OR 853.07  ; 出料伺服Z轴#3腔取料位标志
OR 853.08  ; 出料伺服Z轴#1夹爪氦检NG放料位标志
OR 853.09  ; 出料伺服Z轴#2夹爪氦检NG放料位标志
OR 853.10  ; 出料伺服Z轴#1夹爪配对取放料位标志
OR 853.11  ; 出料伺服Z轴#2夹爪配对取放料位标志
OR W1.00  ; 手动模式
ANDLD
AND P_On
RSET H40.01  ; #2出料夹爪有料记忆
; rung 3
LD H40.01  ; #2出料夹爪有料记忆
OUT 11.00  ; #2出料夹爪夹紧
NOT(520)
AND T0000  ; PLC上电延时100ms
OUT 11.01  ; #2出料夹爪松开

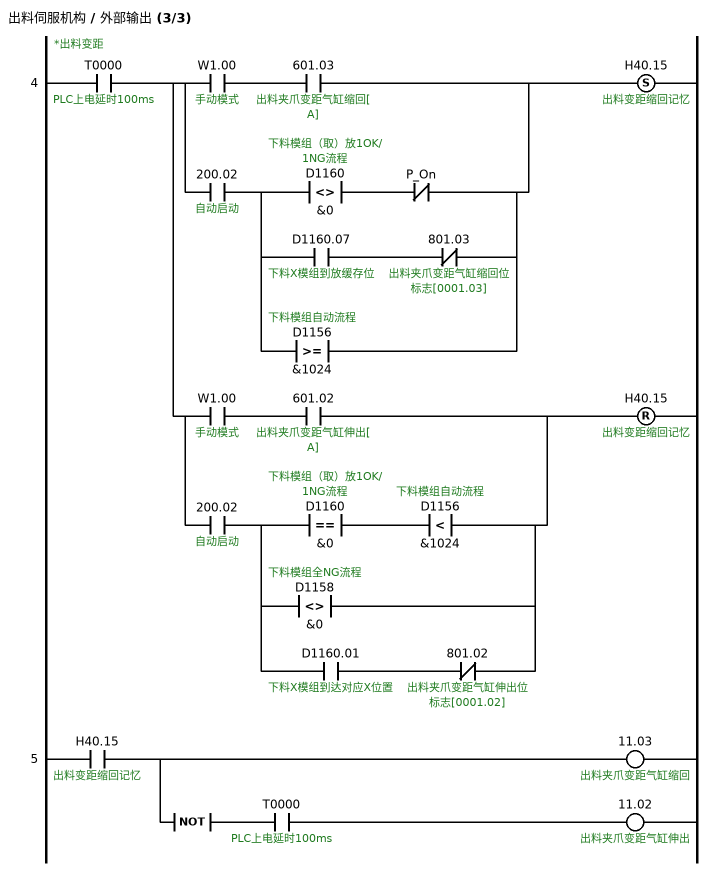
; rung 4: *出料变距
LD T0000  ; PLC上电延时100ms
OUT TR0
LD W1.00  ; 手动模式
AND 601.03  ; 出料夹爪变距气缸缩回[A]
LD 200.02  ; 自动启动
LD<>L(306) D1160 &0  ; 下料模组（取）放1OK/1NG流程
ANDNOT P_On
LD D1160.07  ; 下料X模组到放缓存位
ANDNOT 801.03  ; 出料夹爪变距气缸缩回位标志[0001.03]  // 20190126新增
ORLD
OR>=L(326) D1156 &1024  ; 下料模组自动流程
ANDLD
ORLD
ANDLD
SET H40.15  ; 出料变距缩回记忆
LD TR0
LD W1.00  ; 手动模式
AND 601.02  ; 出料夹爪变距气缸伸出[A]
LD 200.02  ; 自动启动
LD=L(301) D1160 &0  ; 下料模组（取）放1OK/1NG流程
AND<L(311) D1156 &1024  ; 下料模组自动流程
OR<>L(306) D1158 &0  ; 下料模组全NG流程
LD D1160.01  ; 下料X模组到达对应X位置
ANDNOT 801.02  ; 出料夹爪变距气缸伸出位标志[0001.02]  // 20190126新增
ORLD
ANDLD
ORLD
ANDLD
RSET H40.15  ; 出料变距缩回记忆
; rung 5
LD H40.15  ; 出料变距缩回记忆
OUT 11.03  ; 出料夹爪变距气缸缩回
NOT(520)
AND T0000  ; PLC上电延时100ms
OUT 11.02  ; 出料夹爪变距气缸伸出

### Section END
; rung 0
END(001)

## Program NG缓存机构 (cyclic task 5)

### Section NG缓存

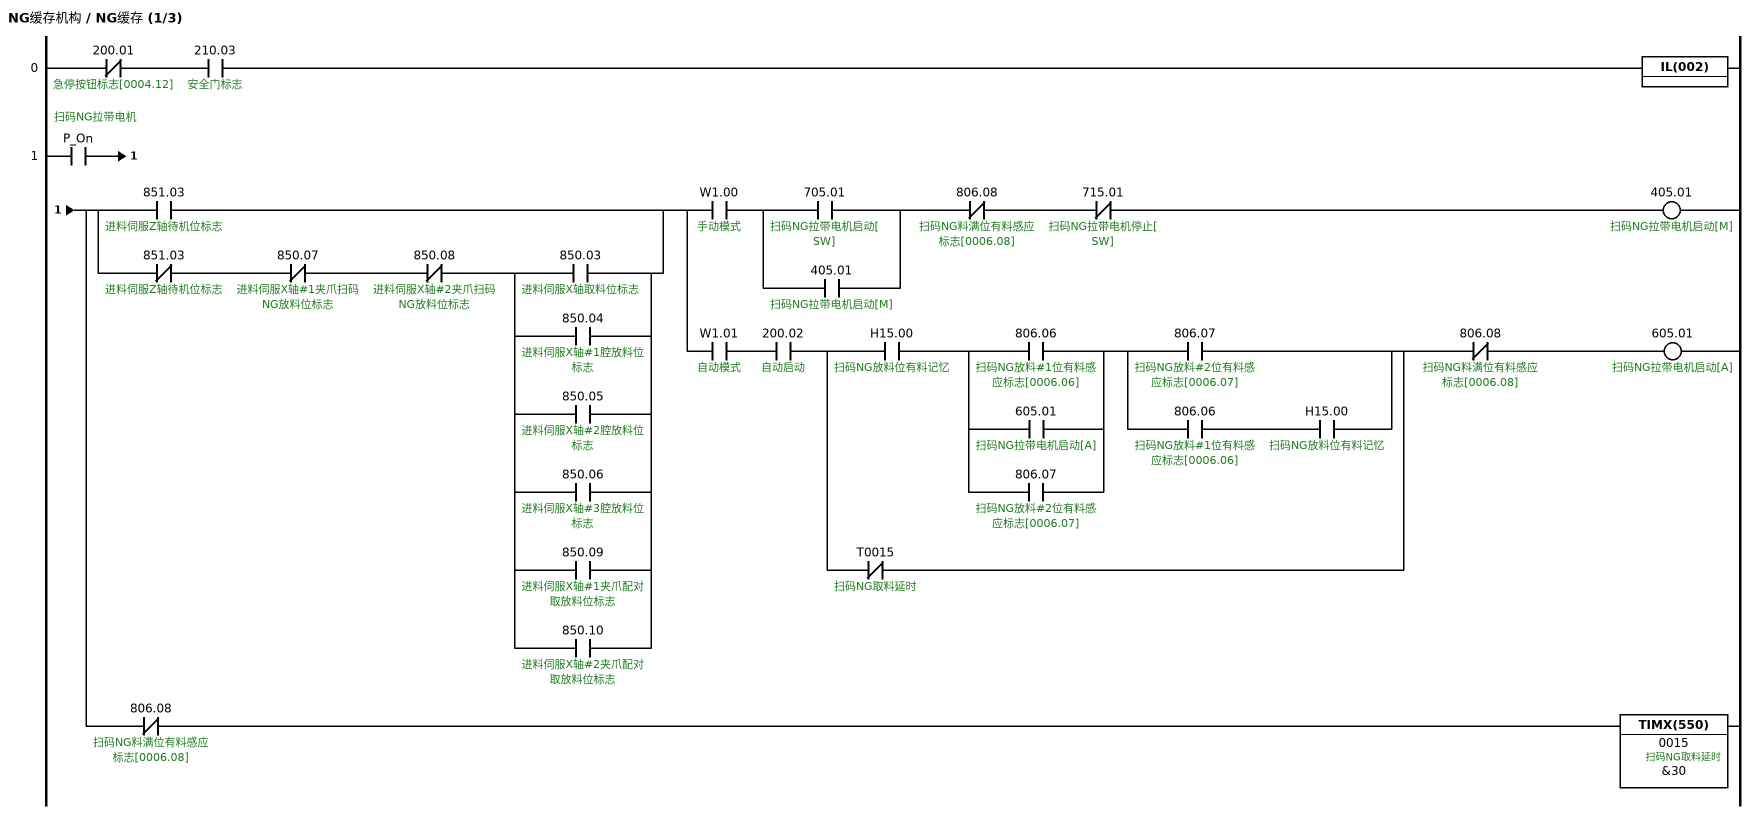
; rung 0
LDNOT 200.01  ; 急停按钮标志[0004.12]
AND 210.03  ; 安全门标志
IL(002)
; rung 1: 扫码NG拉带电机
LD P_On
OUT TR0
LD 851.03  ; 进料伺服Z轴待机位标志
LDNOT 851.03  ; 进料伺服Z轴待机位标志
ANDNOT 850.07  ; 进料伺服X轴#1夹爪扫码NG放料位标志
ANDNOT 850.08  ; 进料伺服X轴#2夹爪扫码NG放料位标志
LD 850.03  ; 进料伺服X轴取料位标志
OR 850.04  ; 进料伺服X轴#1腔放料位标志
OR 850.05  ; 进料伺服X轴#2腔放料位标志
OR 850.06  ; 进料伺服X轴#3腔放料位标志
OR 850.09  ; 进料伺服X轴#1夹爪配对取放料位标志
OR 850.10  ; 进料伺服X轴#2夹爪配对取放料位标志
ANDLD
ORLD
ANDLD
OUT TR1
AND W1.00  ; 手动模式
LD 705.01  ; 扫码NG拉带电机启动[SW]
OR 405.01  ; 扫码NG拉带电机启动[M]
ANDLD
ANDNOT 806.08  ; 扫码NG料满位有料感应标志[0006.08]
ANDNOT 715.01  ; 扫码NG拉带电机停止[SW]
OUT 405.01  ; 扫码NG拉带电机启动[M]
LD TR1
AND W1.01  ; 自动模式
AND 200.02  ; 自动启动
LD H15.00  ; 扫码NG放料位有料记忆
LD 806.06  ; 扫码NG放料#1位有料感应标志[0006.06]
OR 605.01  ; 扫码NG拉带电机启动[A]
OR 806.07  ; 扫码NG放料#2位有料感应标志[0006.07]
ANDLD
LD 806.07  ; 扫码NG放料#2位有料感应标志[0006.07]
LD 806.06  ; 扫码NG放料#1位有料感应标志[0006.06]
AND H15.00  ; 扫码NG放料位有料记忆
ORLD
ANDLD
ORNOT T0015  ; 扫码NG取料延时
ANDLD
ANDNOT 806.08  ; 扫码NG料满位有料感应标志[0006.08]
OUT 605.01  ; 扫码NG拉带电机启动[A]
LD TR0
ANDNOT 806.08  ; 扫码NG料满位有料感应标志[0006.08]
TIMX(550) 0015 &30  ; 扫码NG取料延时

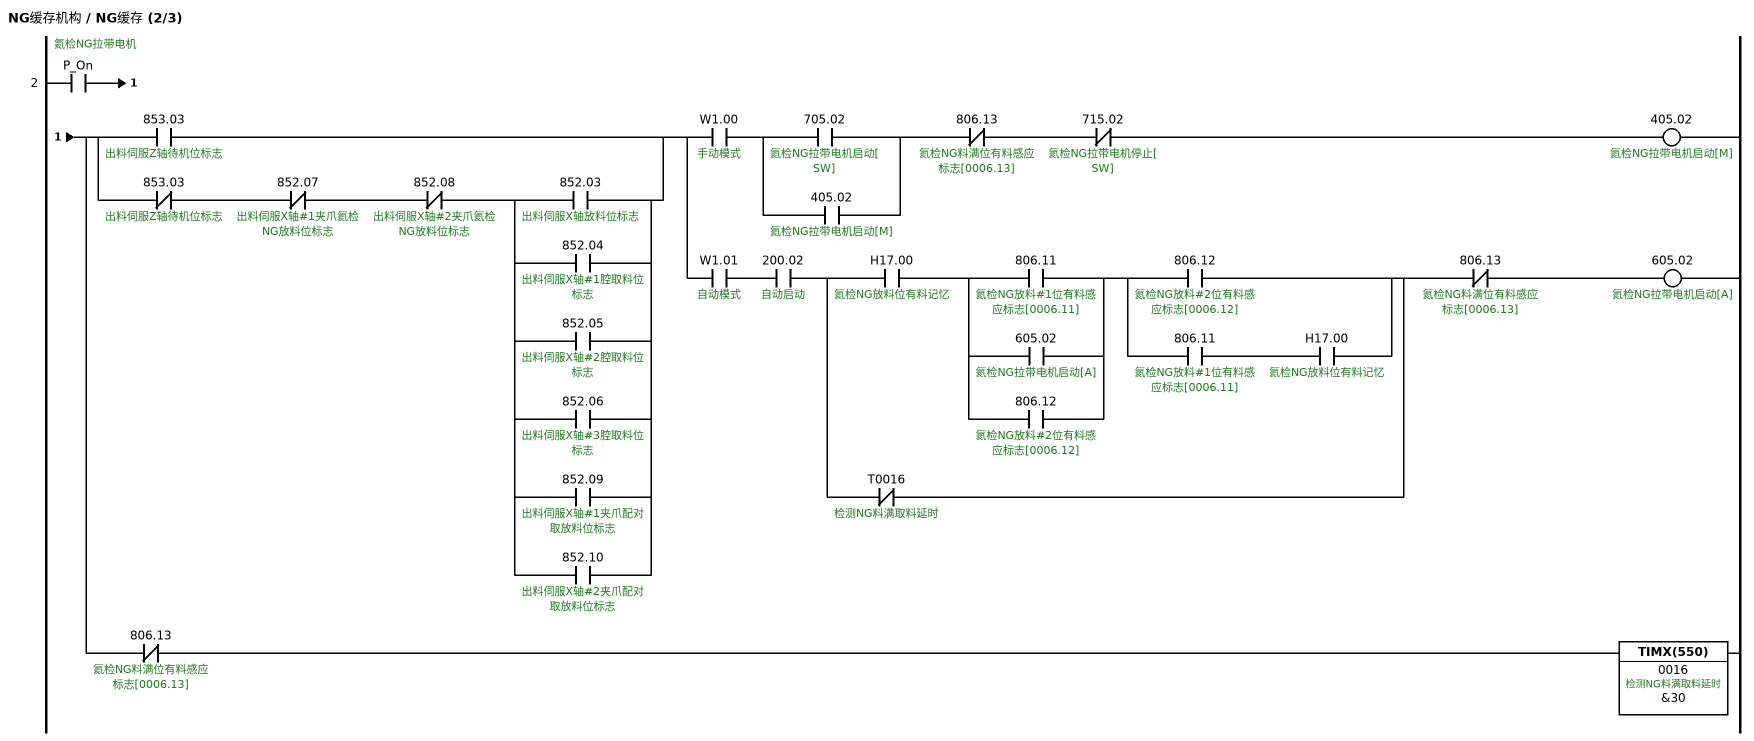
; rung 2: 氦检NG拉带电机
LD P_On
OUT TR0
LD 853.03  ; 出料伺服Z轴待机位标志
LDNOT 853.03  ; 出料伺服Z轴待机位标志
ANDNOT 852.07  ; 出料伺服X轴#1夹爪氦检NG放料位标志
ANDNOT 852.08  ; 出料伺服X轴#2夹爪氦检NG放料位标志
LD 852.03  ; 出料伺服X轴放料位标志
OR 852.04  ; 出料伺服X轴#1腔取料位标志
OR 852.05  ; 出料伺服X轴#2腔取料位标志
OR 852.06  ; 出料伺服X轴#3腔取料位标志
OR 852.09  ; 出料伺服X轴#1夹爪配对取放料位标志
OR 852.10  ; 出料伺服X轴#2夹爪配对取放料位标志
ANDLD
ORLD
ANDLD
OUT TR1
AND W1.00  ; 手动模式
LD 705.02  ; 氦检NG拉带电机启动[SW]
OR 405.02  ; 氦检NG拉带电机启动[M]
ANDLD
ANDNOT 806.13  ; 氦检NG料满位有料感应标志[0006.13]
ANDNOT 715.02  ; 氦检NG拉带电机停止[SW]
OUT 405.02  ; 氦检NG拉带电机启动[M]
LD TR1
AND W1.01  ; 自动模式
AND 200.02  ; 自动启动
LD H17.00  ; 氦检NG放料位有料记忆
LD 806.11  ; 氦检NG放料#1位有料感应标志[0006.11]
OR 605.02  ; 氦检NG拉带电机启动[A]
OR 806.12  ; 氦检NG放料#2位有料感应标志[0006.12]
ANDLD
LD 806.12  ; 氦检NG放料#2位有料感应标志[0006.12]
LD 806.11  ; 氦检NG放料#1位有料感应标志[0006.11]
AND H17.00  ; 氦检NG放料位有料记忆
ORLD
ANDLD
ORNOT T0016  ; 检测NG料满取料延时
ANDLD
ANDNOT 806.13  ; 氦检NG料满位有料感应标志[0006.13]
OUT 605.02  ; 氦检NG拉带电机启动[A]
LD TR0
ANDNOT 806.13  ; 氦检NG料满位有料感应标志[0006.13]
TIMX(550) 0016 &30  ; 检测NG料满取料延时

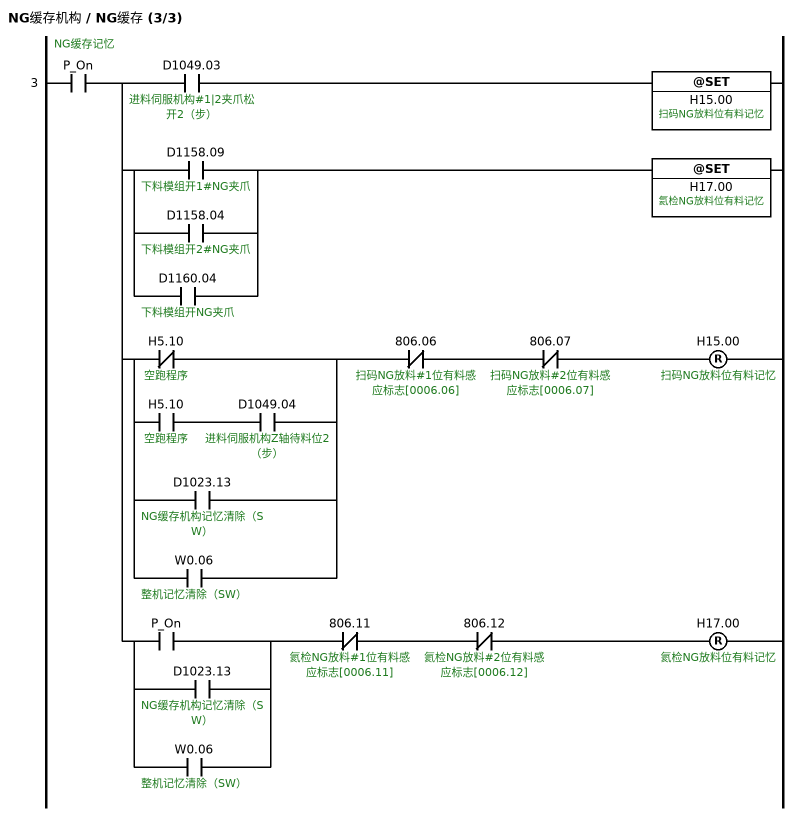
; rung 3: NG缓存记忆
LD P_On
OUT TR0
AND D1049.03  ; 进料伺服机构#1|2夹爪松开2（步）
@SET H15.00  ; 扫码NG放料位有料记忆
LD TR0
LD D1158.09  ; 下料模组开1#NG夹爪
OR D1158.04  ; 下料模组开2#NG夹爪
OR D1160.04  ; 下料模组开NG夹爪
ANDLD
@SET H17.00  ; 氦检NG放料位有料记忆
LD TR0
LDNOT H5.10  ; 空跑程序
LD H5.10  ; 空跑程序
AND D1049.04  ; 进料伺服机构Z轴待料位2（步）
ORLD
OR D1023.13  ; NG缓存机构记忆清除（SW）
OR W0.06  ; 整机记忆清除（SW）
ANDLD
ANDNOT 806.06  ; 扫码NG放料#1位有料感应标志[0006.06]
ANDNOT 806.07  ; 扫码NG放料#2位有料感应标志[0006.07]
RSET H15.00  ; 扫码NG放料位有料记忆
LD TR0
LD P_On
OR D1023.13  ; NG缓存机构记忆清除（SW）
OR W0.06  ; 整机记忆清除（SW）
ANDLD
ANDNOT 806.11  ; 氦检NG放料#1位有料感应标志[0006.11]
ANDNOT 806.12  ; 氦检NG放料#2位有料感应标志[0006.12]
RSET H17.00  ; 氦检NG放料位有料记忆

### Section 外部输出

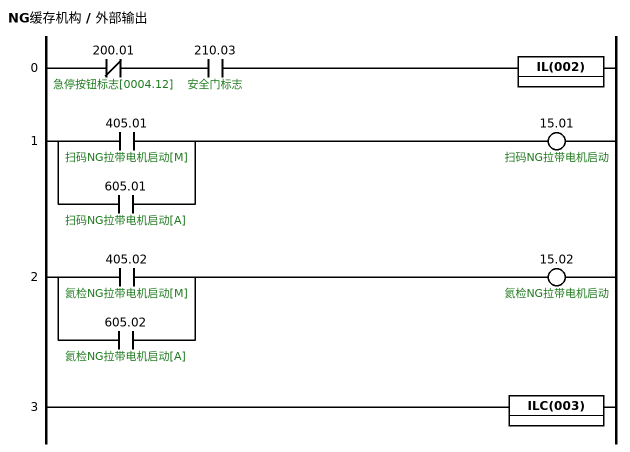
; rung 0
LDNOT 200.01  ; 急停按钮标志[0004.12]
AND 210.03  ; 安全门标志
IL(002)
; rung 1
LD 405.01  ; 扫码NG拉带电机启动[M]
OR 605.01  ; 扫码NG拉带电机启动[A]
OUT 15.01  ; 扫码NG拉带电机启动
; rung 2
LD 405.02  ; 氦检NG拉带电机启动[M]
OR 605.02  ; 氦检NG拉带电机启动[A]
OUT 15.02  ; 氦检NG拉带电机启动
; rung 3
ILC(003)

### Section END
; rung 0
END(001)

## Program Common (cyclic task 6)

### Section 动作延时

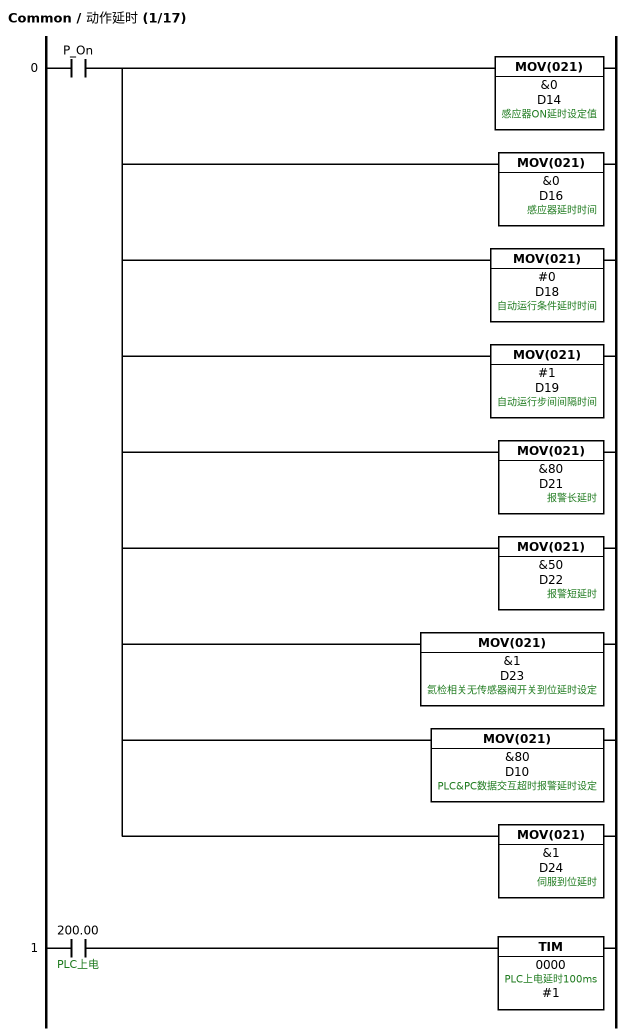
; rung 0
LD P_On
MOV(021) &0 D14  ; 感应器ON延时设定值
MOV(021) &0 D16  ; 感应器延时时间
MOV(021) #0 D18  ; 自动运行条件延时时间
MOV(021) #1 D19  ; 自动运行步间间隔时间
MOV(021) &80 D21  ; 报警长延时
MOV(021) &50 D22  ; 报警短延时
MOV(021) &1 D23  ; 氦检相关无传感器阀开关到位延时设定
MOV(021) &80 D10  ; PLC&PC数据交互超时报警延时设定
MOV(021) &1 D24  ; 伺服到位延时
; rung 1
LD 200.00  ; PLC上电
TIM 0000 #1  ; PLC上电延时100ms

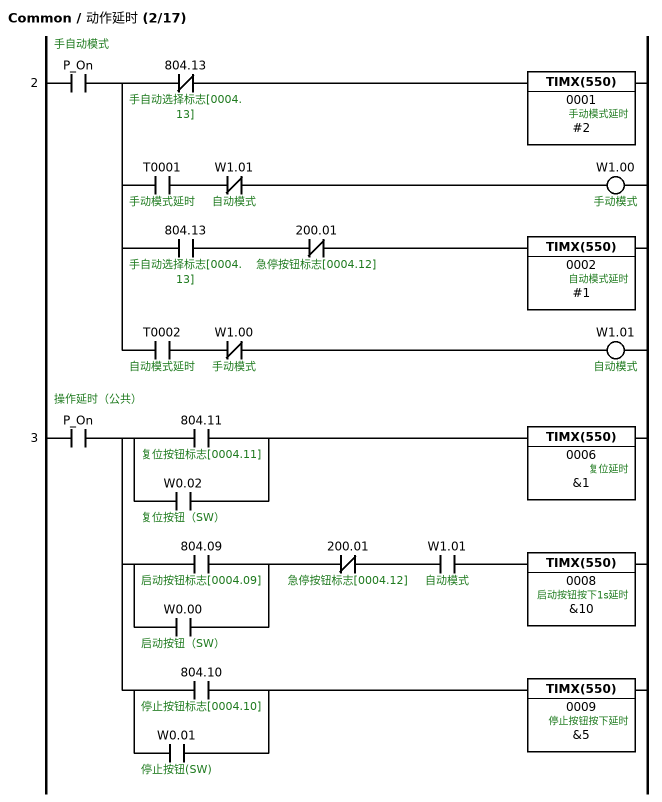
; rung 2: 手自动模式
LD P_On
OUT TR0
ANDNOT 804.13  ; 手自动选择标志[0004.13]
TIMX(550) 0001 #2  ; 手动模式延时
LD TR0
AND T0001  ; 手动模式延时
ANDNOT W1.01  ; 自动模式
OUT W1.00  ; 手动模式
LD TR0
AND 804.13  ; 手自动选择标志[0004.13]
ANDNOT 200.01  ; 急停按钮标志[0004.12]
TIMX(550) 0002 #1  ; 自动模式延时
LD TR0
AND T0002  ; 自动模式延时
ANDNOT W1.00  ; 手动模式
OUT W1.01  ; 自动模式
; rung 3: 操作延时（公共）
LD P_On
OUT TR0
LD 804.11  ; 复位按钮标志[0004.11]
OR W0.02  ; 复位按钮（SW）
ANDLD
TIMX(550) 0006 &1  ; 复位延时
LD TR0
LD 804.09  ; 启动按钮标志[0004.09]
OR W0.00  ; 启动按钮（SW）
ANDLD
ANDNOT 200.01  ; 急停按钮标志[0004.12]
AND W1.01  ; 自动模式
TIMX(550) 0008 &10  ; 启动按钮按下1s延时
LD TR0
LD 804.10  ; 停止按钮标志[0004.10]
OR W0.01  ; 停止按钮(SW)
ANDLD
TIMX(550) 0009 &5  ; 停止按钮按下延时

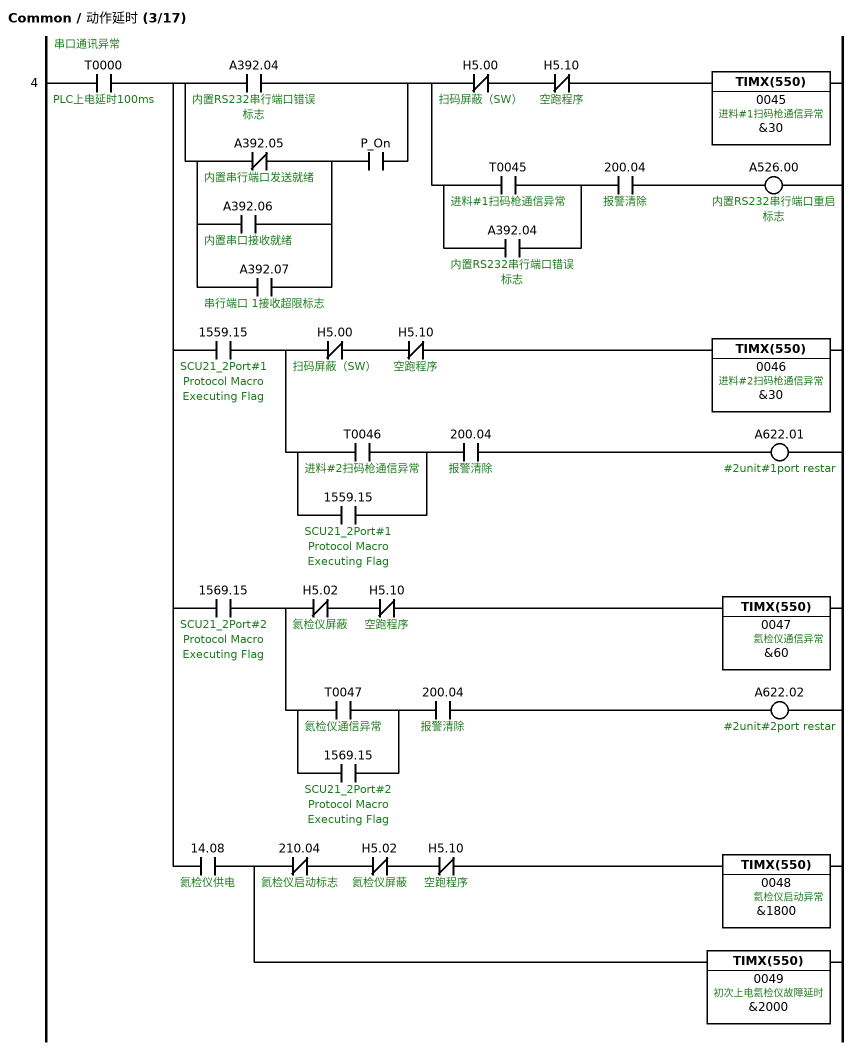
; rung 4: 串口通讯异常
LD T0000  ; PLC上电延时100ms
OUT TR0
LD A392.04  ; 内置RS232串行端口错误标志
LDNOT A392.05  ; 内置串行端口发送就绪
OR A392.06  ; 内置串口接收就绪
OR A392.07  ; 串行端口 1接收超限标志
AND P_On
ORLD
ANDLD
OUT TR1
ANDNOT H5.00  ; 扫码屏蔽（SW）
ANDNOT H5.10  ; 空跑程序
TIMX(550) 0045 &30  ; 进料#1扫码枪通信异常
LD TR1
LD T0045  ; 进料#1扫码枪通信异常
OR A392.04  ; 内置RS232串行端口错误标志
ANDLD
AND 200.04  ; 报警清除
OUT A526.00  ; 内置RS232串行端口重启标志
LD TR0
AND 1559.15  ; SCU21_2Port#1 Protocol Macro Executing Flag
OUT TR1
ANDNOT H5.00  ; 扫码屏蔽（SW）
ANDNOT H5.10  ; 空跑程序
TIMX(550) 0046 &30  ; 进料#2扫码枪通信异常
LD TR1
LD T0046  ; 进料#2扫码枪通信异常
OR 1559.15  ; SCU21_2Port#1 Protocol Macro Executing Flag
ANDLD
AND 200.04  ; 报警清除
OUT A622.01  ; #2unit#1port restar
LD TR0
AND 1569.15  ; SCU21_2Port#2 Protocol Macro Executing Flag
OUT TR1
ANDNOT H5.02  ; 氦检仪屏蔽
ANDNOT H5.10  ; 空跑程序
TIMX(550) 0047 &60  ; 氦检仪通信异常
LD TR1
LD T0047  ; 氦检仪通信异常
OR 1569.15  ; SCU21_2Port#2 Protocol Macro Executing Flag
ANDLD
AND 200.04  ; 报警清除
OUT A622.02  ; #2unit#2port restar
LD TR0
AND 14.08  ; 氦检仪供电
OUT TR0
ANDNOT 210.04  ; 氦检仪启动标志
ANDNOT H5.02  ; 氦检仪屏蔽
ANDNOT H5.10  ; 空跑程序
TIMX(550) 0048 &1800  ; 氦检仪启动异常
LD TR0
TIMX(550) 0049 &2000  ; 初次上电氦检仪故障延时
; rung 5: AI断线检测

